FUNCTION GetMaterialLengthFromCode : INT
VAR_INPUT
	materialID : STRING;
END_VAR
VAR
	temp : STRING;
	getNumFromString : FB_EnumStringNumbers;
END_VAR

getNumFromString(
	sSearch:= materialID, 
	eCmd:= eEnumCmd_First, 
	eType:= eNumGroup_Unsigned, 
	sNumber=> temp, 
	nPos=> , 
	bEOS=> );
	
GetMaterialLengthFromCode := TO_INT(TO_INT(temp) * 25.4); //inch to mm

END_FUNCTION

(* stored: Version 1.1.0.1, ProductVersion 3.1.4024.11
   POU GetMaterialLengthFromCode: Id {8bc76473-7909-4f63-aec3-56c20496ed83}, SpecialFunc None *)
